PROGRAM PRG_Test
VAR
	fb_VGC_Test: FB_VGC_Test;
	fb_VRC_Test: FB_VRC_Test;
	fb_PIP_Test: FB_PIP_Test;
	fb_PTM_Test: FB_PTM_Test;
	fb_GPI_Test:FB_GPI_Test;
	fb_GCC_Test:FB_GCC_Test;

	TotalTests : INT:=0;
END_VAR


TcUnit.RUN();

END_PROGRAM

(* stored: Version 1.1.0.1, ProductVersion 3.1.4022.18
   POU PRG_Test: Id {3d3ce199-d6e8-49d3-9e69-49f0a2678e11}, SpecialFunc None *)
